// TIA Portal V21 export
ORGANIZATION_BLOCK "Main"   // OB1, LAD, ProgramCycle
TITLE = "Main Program Sweep (Cycle)"
{ S7_Optimized_Access := 'TRUE' }
// stored: SetENOAutomatically false
   VAR_INPUT
      Initial_Call : Bool;   // Initial call of this OB
      Remanence : Bool;   // =True, if remanent data are available
   END_VAR
BEGIN

REGION Network 1: Cabinet management
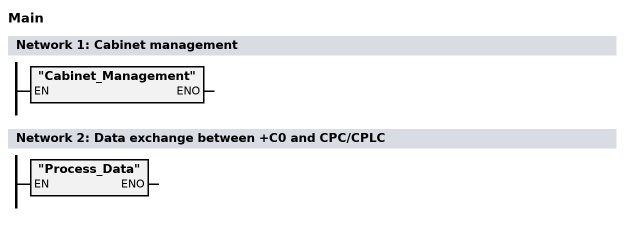
   RUNG wire#powerrail
      "Cabinet_Management"()
   END_RUNG
   // the same network as SCL:
   "Cabinet_Management"();
END_REGION

REGION Network 2: Data exchange between +C0 and CPC/CPLC
   RUNG wire#powerrail
      "Process_Data"()
   END_RUNG
   // the same network as SCL:
   "Process_Data"();
END_REGION
END_ORGANIZATION_BLOCK
